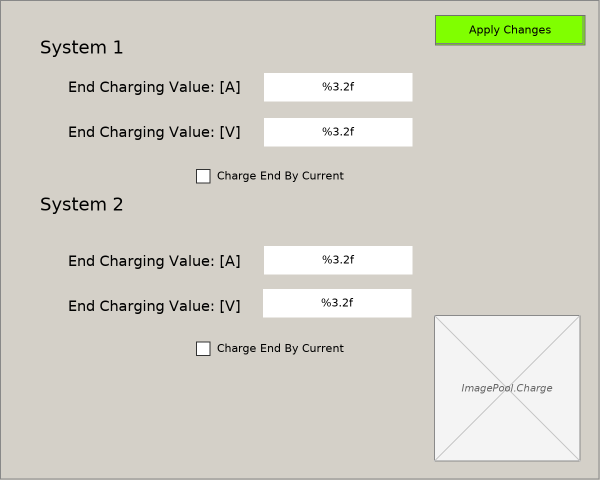
VISUALIZATION vCharging  // 600x480
    Label (28,35 108x25), "System 1"
    Label (28,192 108x25), "System 2"
    Textfield (263,72 150x30), "%3.2f", text variable: ACTION1.rEndCharginValue
        OnMouseClick: write the text variable via Default
    Label (54,72 201x30), "End Charging Value: [A]"
    Textfield (263,245 150x30), "%3.2f", text variable: ACTION2.rEndCharginValue
        OnMouseClick: write the text variable via Default
    Button (435,15 150x30), "Apply Changes"
        OnMouseClick: execute { MAIN.bSetPerData:=true; }
    Image (434,315 146x146), image: ImagePool.Charge
    Textfield (262,288 150x30), "%3.2f", text variable: ACTION2.rEndCharginValueVoltage
        OnMouseClick: write the text variable via Default
    Textfield (263,117 150x30), "%3.2f", text variable: ACTION1.rEndCharginValueVoltage
        OnMouseClick: write the text variable via Default
    Label (54,117 201x30), "End Charging Value: [V]"
    Checkbox (194,158 167x36), "Charge End By Current", variable: ACTION1.bChargingByCurrent, input disabled if: false
    Checkbox (194,331 167x35), "Charge End By Current", variable: ACTION2.bChargingByCurrent, input disabled if: false
    Label (54,246 201x30), "End Charging Value: [A]"
    Label (54,291 201x30), "End Charging Value: [V]"
END_VISUALIZATION

(* stored: Version 1.1.0.1, ProductVersion 3.1.4024.12
   Visu vCharging: Id {c8171bee-7cfe-4cf6-9ca1-1ba77733a947} *)
